(* Logix 5000 project; controller PLCbox vendor 1 type 14 code 149 rev 30.11; software revision 30.01; part 2 of 4 *)
(* tags used below, declared in another part *)
   CurrentRecipe : DINT;
   Recipe : DINT[10];
   ValveBank2 : BOOL[32];
   AnalogInput : REAL[100];
   AnalogScaled : REAL[100];
   BoxCounter : COUNTER;
   IN_Loc1 : BOOL[32];
   IN_Loc1_DB_OFF : BOOL[32];
   IN_Loc1_DB_ON : BOOL[32];
   IN_Loc1_Index : DINT;
   IN_Loc1_T_OFF : TIMER[16];
   IN_Loc1_T_ON : TIMER[16];
   LocalOut : DINT[20];
   OUT_Loc1 : BOOL[32];
   PID_Analog_In : REAL[20];
   PLCTime : UDT_Time;
   SsytemStopped : BOOL;
(* InterviewPractice, continued *)

ROUTINE _03_MEQrecipe   (* ladder *)
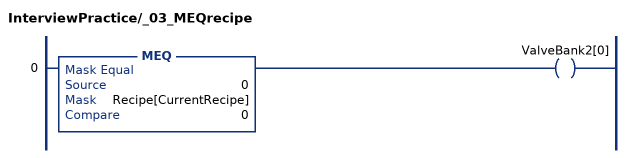
   0: MEQ(0,Recipe[CurrentRecipe],0)OTE(ValveBank2[0]);
END_ROUTINE
END_PROGRAM

PROGRAM JumpTest   (* main routine _01_Main *)
VAR
   Local : BOOL[64] := ([0] := 1, [1] := 1);
END_VAR

ROUTINE _01_Main   (* ladder *)
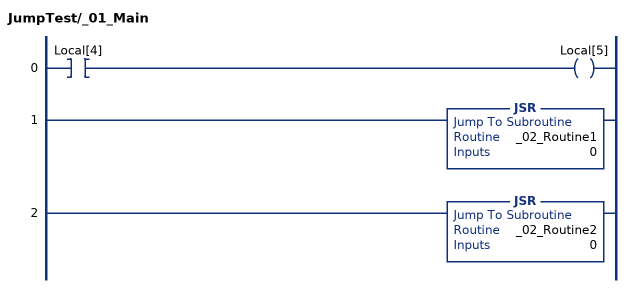
   0: XIC(Local[4])OTE(Local[5]);
   1: JSR(_02_Routine1,0);
   2: JSR(_02_Routine2,0);
END_ROUTINE

ROUTINE _02_Routine1   (* ladder *)
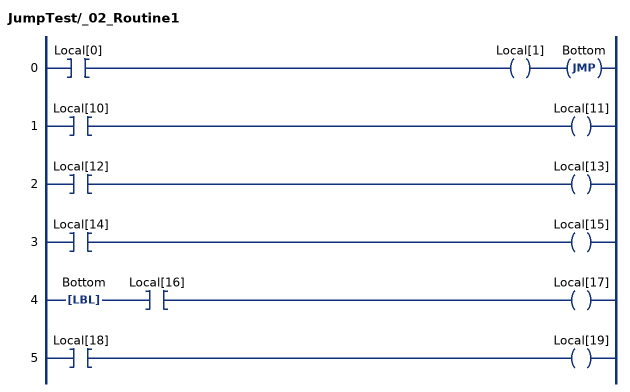
   0: XIC(Local[0])OTE(Local[1])JMP(Bottom);
   1: XIC(Local[10])OTE(Local[11]);
   2: XIC(Local[12])OTE(Local[13]);
   3: XIC(Local[14])OTE(Local[15]);
   4: LBL(Bottom)XIC(Local[16])OTE(Local[17]);
   5: XIC(Local[18])OTE(Local[19]);
END_ROUTINE

ROUTINE _02_Routine2   (* ladder *)
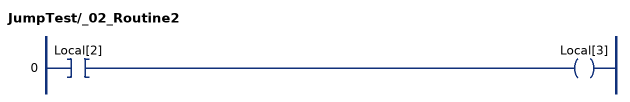
   0: XIC(Local[2])OTE(Local[3]);
END_ROUTINE
END_PROGRAM

PROGRAM MainProgram   (* main routine _01_Main *)
VAR
   ClearString : String20;
   FinalCode : String20 := '$00$00$00$00$00$00$00$00$00$00$00$00$C4$016$F1$00$00$00$00';
   Input_Tag : BOOL := 1;
   LocalDebounceTimer : TIMER;
   LocInDebounced1 : BOOL;
   MFinalCode : String20 := 'VW$00$00$00$00$00$00$1C$00$00$80$C4$016$F1$00$00$00$00';
   MyBarcode : STRING := '$00$00$00$00$00$00$00$00$00$00$00$00$C4$016$F1$00$00$00$00$CE$8F$0A$00X$00$00$0063013337$0A$00$00$80$1C$00$00$80$C4$016$F1$00$00$00$00$CE$8F$0A$00X$00$00$0063013337$0A$00$00$80$1C$00$00$80$C4$016$F1$00$00$00$00';
   OUT_Loc1_AUTO : BOOL[32] := ([0] := 1, [1] := 1, [2] := 1, [3] := 1, [4] := 1, [5] := 1, [6] := 1, [7] := 1, [8] := 1, [9] := 1, [10] := 1, [11] := 1, [12] := 1, [13] := 1, [14] := 1, [15] := 1, [16] := 1, [17] := 1, [18] := 1, [19] := 1, [20] := 1, [21] := 1, [22] := 1, [23] := 1, [24] := 1, [25] := 1, [26] := 1, [27] := 1, [28] := 1, [29] := 1, [30] := 1, [31] := 1);
   OUT_Loc1_F : BOOL[32] := ([0] := 1, [1] := 1);
   OUT_Loc1_Final : BOOL;
   OUT_Loc1_FORCE : BOOL[32];
   OUT_Loc1_Index : DINT := 16;
   OUT_S1 : UDT_Output[16] := ([0].Auto := 1, [0].ManualAvl := 1, [0].Force := 1, [0].Name := 'Test Tag', [1].ManualAvl := 1, [1].Force := 1, [1].ForceAvl := 1, [2].Auto := 1, [2].ManualAvl := 1, [3].ManualAvl := 1, [3].ForceAvl := 1, [4].Auto := 1, [4].ManualAvl := 1, [5].ManualAvl := 1, [5].ForceAvl := 1, [6].ManualAvl := 1, [6].ForceAvl := 1, [7].ManualAvl := 1, [7].ForceAvl := 1, [8].ManualAvl := 1, [8].ForceAvl := 1, [9].Auto := 1, [9].ManualAvl := 1, [10].Auto := 1, [10].ManualAvl := 1, [11].ManualAvl := 1, [11].ForceAvl := 1, [12].ManualAvl := 1, [12].ForceAvl := 1, [13].ManualAvl := 1, [13].ForceAvl := 1, [14].ManualAvl := 1, [14].ForceAvl := 1, [15].ManualAvl := 1, [15].ForceAvl := 1);
   Output_Tag : BOOL;
   SCL_01 : SCALE;
   STR : STRING := '825242422';
   test : DINT := 825242422;
   test2 : DINT[2];
END_VAR

ROUTINE _01_Main   (* ladder *)
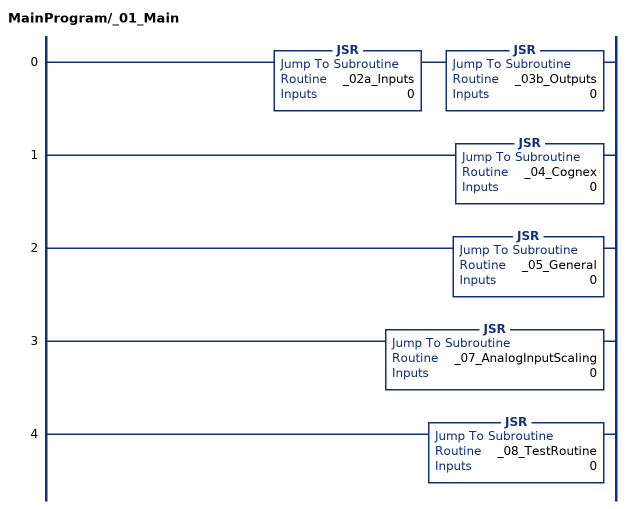
   0: JSR(_02a_Inputs,0)JSR(_03b_Outputs,0);
   1: JSR(_04_Cognex,0);
   2: JSR(_05_General,0);
   3: JSR(_07_AnalogInputScaling,0);
   4: JSR(_08_TestRoutine,0);
END_ROUTINE

ROUTINE _02a_Inputs   (* ladder *)
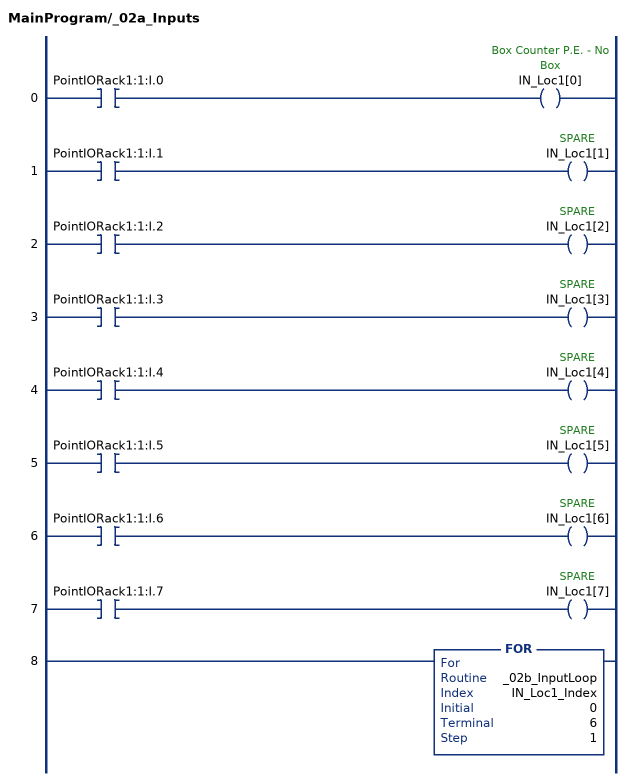
   0: XIC(PointIORack1:1:I.0)OTE(IN_Loc1[0]);
   1: XIC(PointIORack1:1:I.1)OTE(IN_Loc1[1]);
   2: XIC(PointIORack1:1:I.2)OTE(IN_Loc1[2]);
   3: XIC(PointIORack1:1:I.3)OTE(IN_Loc1[3]);
   4: XIC(PointIORack1:1:I.4)OTE(IN_Loc1[4]);
   5: XIC(PointIORack1:1:I.5)OTE(IN_Loc1[5]);
   6: XIC(PointIORack1:1:I.6)OTE(IN_Loc1[6]);
   7: XIC(PointIORack1:1:I.7)OTE(IN_Loc1[7]);
   8: FOR(_02b_InputLoop,IN_Loc1_Index,0,6,1);
END_ROUTINE

ROUTINE _02b_InputLoop   (* ladder *)
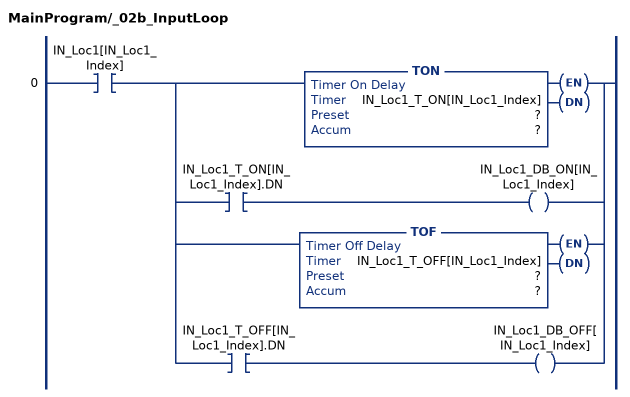
   0: XIC(IN_Loc1[IN_Loc1_Index])[TON(IN_Loc1_T_ON[IN_Loc1_Index],?,?) ,XIC(IN_Loc1_T_ON[IN_Loc1_Index].DN) OTE(IN_Loc1_DB_ON[IN_Loc1_Index]) ,TOF(IN_Loc1_T_OFF[IN_Loc1_Index],?,?) ,XIC(IN_Loc1_T_OFF[IN_Loc1_Index].DN) OTE(IN_Loc1_DB_OFF[IN_Loc1_Index]) ];
END_ROUTINE

ROUTINE _03a_Outputs   (* ladder *)
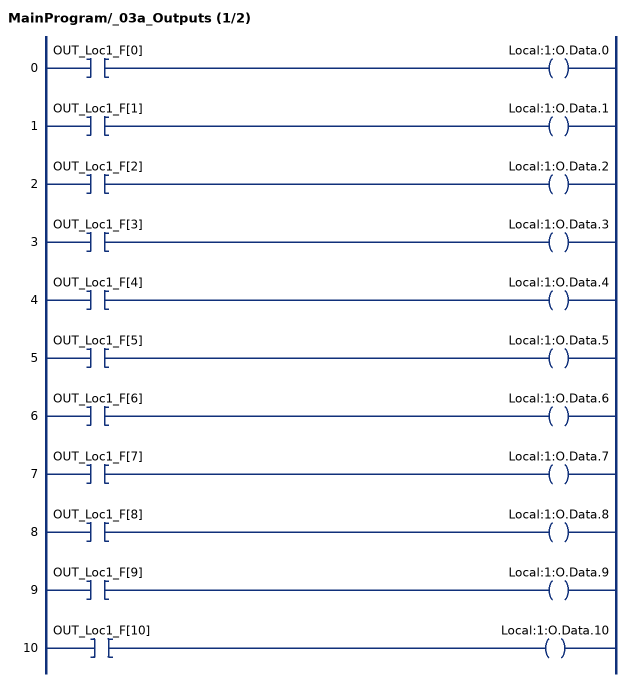
   0: XIC(OUT_Loc1_F[0])OTE(Local:1:O.Data.0);
   1: XIC(OUT_Loc1_F[1])OTE(Local:1:O.Data.1);
   2: XIC(OUT_Loc1_F[2])OTE(Local:1:O.Data.2);
   3: XIC(OUT_Loc1_F[3])OTE(Local:1:O.Data.3);
   4: XIC(OUT_Loc1_F[4])OTE(Local:1:O.Data.4);
   5: XIC(OUT_Loc1_F[5])OTE(Local:1:O.Data.5);
   6: XIC(OUT_Loc1_F[6])OTE(Local:1:O.Data.6);
   7: XIC(OUT_Loc1_F[7])OTE(Local:1:O.Data.7);
   8: XIC(OUT_Loc1_F[8])OTE(Local:1:O.Data.8);
   9: XIC(OUT_Loc1_F[9])OTE(Local:1:O.Data.9);
   10: XIC(OUT_Loc1_F[10])OTE(Local:1:O.Data.10);
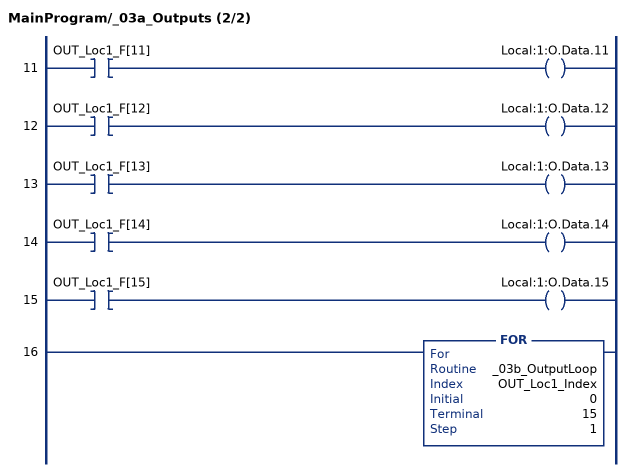
   11: XIC(OUT_Loc1_F[11])OTE(Local:1:O.Data.11);
   12: XIC(OUT_Loc1_F[12])OTE(Local:1:O.Data.12);
   13: XIC(OUT_Loc1_F[13])OTE(Local:1:O.Data.13);
   14: XIC(OUT_Loc1_F[14])OTE(Local:1:O.Data.14);
   15: XIC(OUT_Loc1_F[15])OTE(Local:1:O.Data.15);
   16: FOR(_03b_OutputLoop,OUT_Loc1_Index,0,15,1);
END_ROUTINE

ROUTINE _03b_OutputLoop   (* ladder *)
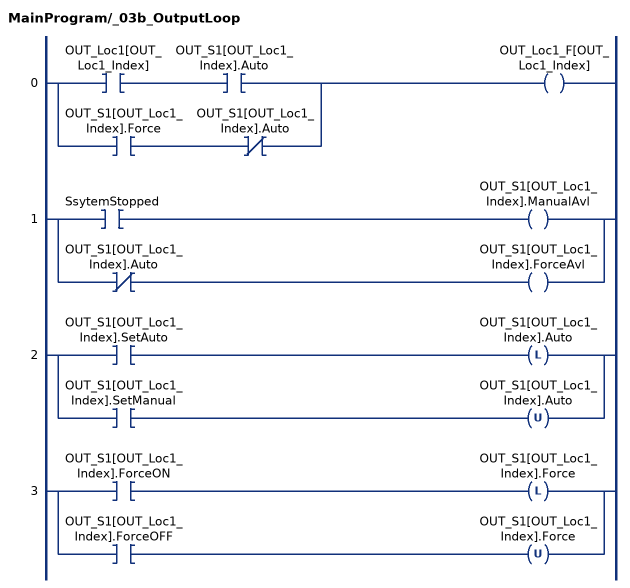
   0: [XIC(OUT_Loc1[OUT_Loc1_Index]) XIC(OUT_S1[OUT_Loc1_Index].Auto) ,XIC(OUT_S1[OUT_Loc1_Index].Force) XIO(OUT_S1[OUT_Loc1_Index].Auto) ]OTE(OUT_Loc1_F[OUT_Loc1_Index]);
   1: [XIC(SsytemStopped) OTE(OUT_S1[OUT_Loc1_Index].ManualAvl) ,XIO(OUT_S1[OUT_Loc1_Index].Auto) OTE(OUT_S1[OUT_Loc1_Index].ForceAvl) ];
   2: [XIC(OUT_S1[OUT_Loc1_Index].SetAuto) OTL(OUT_S1[OUT_Loc1_Index].Auto) ,XIC(OUT_S1[OUT_Loc1_Index].SetManual) OTU(OUT_S1[OUT_Loc1_Index].Auto) ];
   3: [XIC(OUT_S1[OUT_Loc1_Index].ForceON) OTL(OUT_S1[OUT_Loc1_Index].Force) ,XIC(OUT_S1[OUT_Loc1_Index].ForceOFF) OTU(OUT_S1[OUT_Loc1_Index].Force) ];
END_ROUTINE

ROUTINE _03b_Outputs   (* structured text *)
   Local:1:O.Data.0 [:=] LocalOut[2].0; //E-Stop LED Light
   Local:1:O.Data.1 [:=] LocalOut[2].1; //System Ready LED Light
   Local:1:O.Data.2 [:=] LocalOut[2].2; //Case Packer Ready Signal
   Local:1:O.Data.3 [:=] LocalOut[2].3; //Case Packer Faulted Signal
   Local:1:O.Data.4 [:=] LocalOut[2].4; //MTR3005
   Local:1:O.Data.5 [:=] LocalOut[2].5; //SPARE
   Local:1:O.Data.6 [:=] LocalOut[2].6; //SPARE
   Local:1:O.Data.7 [:=] LocalOut[2].7; //SPARE
   Local:1:O.Data.8 [:=] LocalOut[2].8; //SPARE
   Local:1:O.Data.9 [:=] LocalOut[2].9; //SPARE
   Local:1:O.Data.10 [:=] LocalOut[2].10; //SPARE
   Local:1:O.Data.11 [:=] LocalOut[2].11; //SPARE
   Local:1:O.Data.12 [:=] LocalOut[2].12; //SPARE
   Local:1:O.Data.13 [:=] LocalOut[2].13; //SPARE
   Local:1:O.Data.14 [:=] LocalOut[2].14; //SPARE
   Local:1:O.Data.15 [:=] LocalOut[2].15; //SPARE
END_ROUTINE

ROUTINE _04_Cognex   (* ladder *)
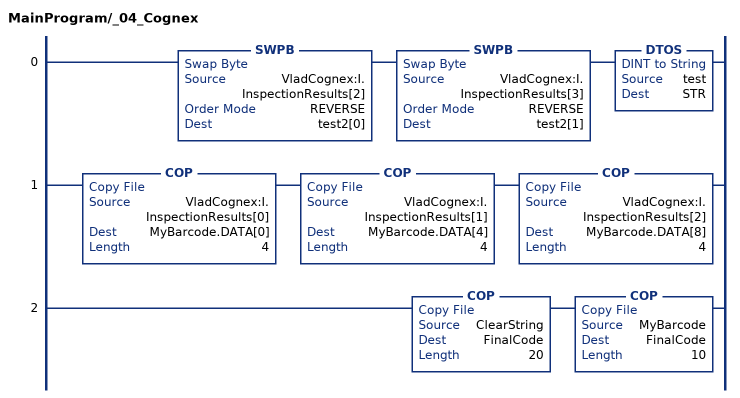
   0: SWPB(VladCognex:I.InspectionResults[2],REVERSE,test2[0])SWPB(VladCognex:I.InspectionResults[3],REVERSE,test2[1])DTOS(test,STR);
   1: COP(VladCognex:I.InspectionResults[0],MyBarcode.DATA[0],4)COP(VladCognex:I.InspectionResults[1],MyBarcode.DATA[4],4)COP(VladCognex:I.InspectionResults[2],MyBarcode.DATA[8],4);
   2: COP(ClearString,FinalCode,20)COP(MyBarcode,FinalCode,10);
END_ROUTINE

ROUTINE _05_General   (* ladder *)
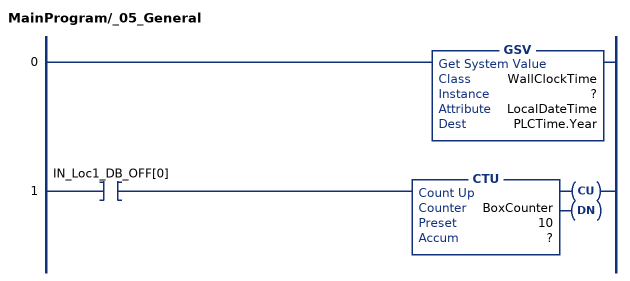
   0: GSV(WallClockTime,?,LocalDateTime,PLCTime.Year);
   1: XIC(IN_Loc1_DB_OFF[0])CTU(BoxCounter,?,?);
END_ROUTINE

ROUTINE _06_Ext_Inputs   (* ladder *)
END_ROUTINE

ROUTINE _07_AnalogInputScaling   (* function block diagram *)
   SHEET 1
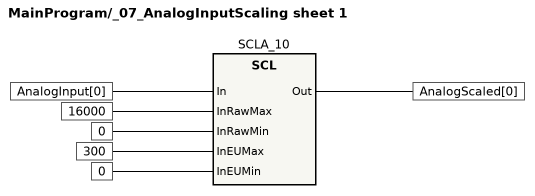
   SCLA_10 : SCL(In := AnalogInput[0], InRawMax := 16000, InRawMin := 0, InEUMax := 300, InEUMin := 0);
   AnalogScaled[0] := SCLA_10.Out;
END_ROUTINE

ROUTINE _08_TestRoutine   (* ladder *)
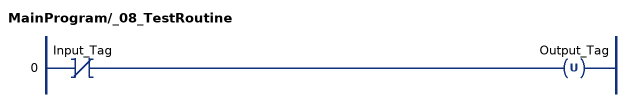
   0: XIO(Input_Tag)OTU(Output_Tag);
END_ROUTINE
END_PROGRAM

PROGRAM MainProgram2   (* main routine _01_Main *)
VAR
   PID_1001 : PID_ENHANCED := (PVEUMax := 100.0, SPOper := 50.0, SPHLimit := 100.0, RatioProg := 1.0, RatioOper := 1.0, RatioHLimit := 1.0, RatioLLimit := 1.0, CVOper := 100.0, CVEUMax := 100.0, CVHLimit := 100.0, DependIndepend := 1, PGain := 0.1, IGain := 0.001, DGain := 0.001, PVEDerivative := 1, ProgOperReq := 1, RTSTime := 1, CVEU := 100.0, CV := 100.0, CVHAlarm := 1, SP := 50.0, SPPercent := 50.0, E := 50.0, EPercent := 50.0, InitPrimary := 1, WindupHOut := 1, Ratio := 1.0, Auto := 1, DeltaT := 0.1);
   PID_Par_1001 : UDT_PID := (P := 0.1, I := 0.001, D := 0.001, CV := 100.0, SP := 50.0, Auto := 1, Name := 'PID 1001 - Testing CLICK PLC Input');
   SCL_01 : SCALE := (InRawMax := 5000.0, InEUMax := 100.0);
END_VAR

ROUTINE _01_Main   (* ladder *)
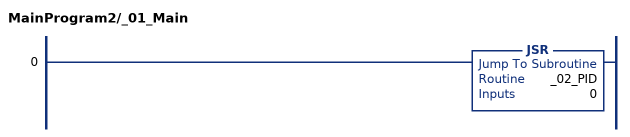
   0: JSR(_02_PID,0);
END_ROUTINE

ROUTINE _02_PID   (* function block diagram *)
   SHEET 1
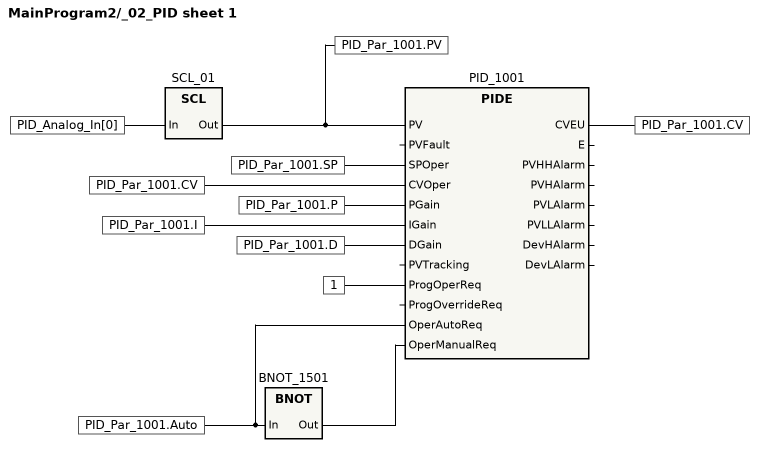
   SCL_01 : SCL(In := PID_Analog_In[0]);
   BNOT_1501 : BNOT(In := PID_Par_1001.Auto);
   PID_Par_1001.PV := SCL_01.Out;
   PID_1001 : PIDE(PV := SCL_01.Out, SPOper := PID_Par_1001.SP, CVOper := PID_Par_1001.CV, PGain := PID_Par_1001.P, IGain := PID_Par_1001.I, DGain := PID_Par_1001.D, ProgOperReq := 1, OperAutoReq := PID_Par_1001.Auto, OperManualReq := BNOT_1501.Out);   // unwired pins: PVFault PVTracking ProgOverrideReq E PVHHAlarm PVHAlarm PVLAlarm PVLLAlarm DevHAlarm DevLAlarm
   PID_Par_1001.CV := PID_1001.CVEU;
END_ROUTINE
END_PROGRAM

PROGRAM Mathematical   (* main routine _01_Main *)
VAR
   System_DINT : DINT[100] := ([0] := 12, [1] := 32, [2] := 54, [3] := 4, [4] := 31, [5] := 38, [6] := 100, [7] := 50, [8] := 200, [9] := 116);
   System_REAL : REAL[100] := ([0] := 23.0, [1] := 42.0, [2] := 0.48835304, [5] := 1.0);
END_VAR

ROUTINE _01_Main   (* ladder *)
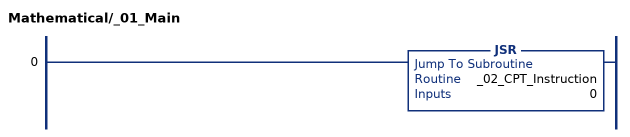
   0: JSR(_02_CPT_Instruction,0);
END_ROUTINE

ROUTINE _02_CPT_Instruction   (* ladder *)
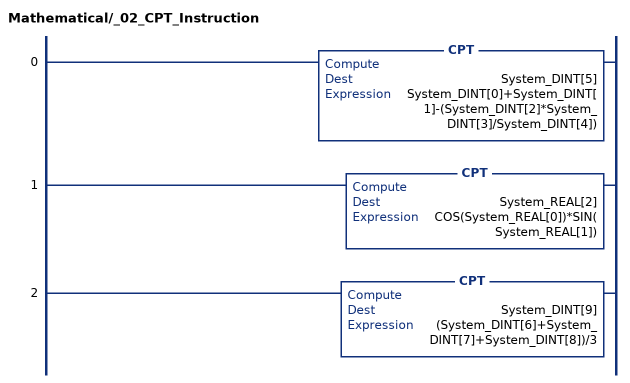
   0: CPT(System_DINT[5],System_DINT[0]+System_DINT[1]-(System_DINT[2]*System_DINT[3]/System_DINT[4]));
   1: CPT(System_REAL[2],COS(System_REAL[0])*SIN(System_REAL[1]));
   2: CPT(System_DINT[9],(System_DINT[6]+System_DINT[7]+System_DINT[8])/3);
END_ROUTINE
END_PROGRAM
